FUNCTION_BLOCK PUBLIC POU_blank_FB
VAR_INPUT
END_VAR
VAR_OUTPUT
END_VAR
VAR
END_VAR

END_FUNCTION_BLOCK

(* stored: Version 1.1.0.1, ProductVersion 3.1.4022.6
   POU POU_blank_FB: Id {06fdbe19-e246-445b-aa76-3d223c3c40af}, SpecialFunc None *)
